// Mitsubishi GX Works2 project: 선입우선회로   PLC: Q02/Q02H

PROGRAM MAIN
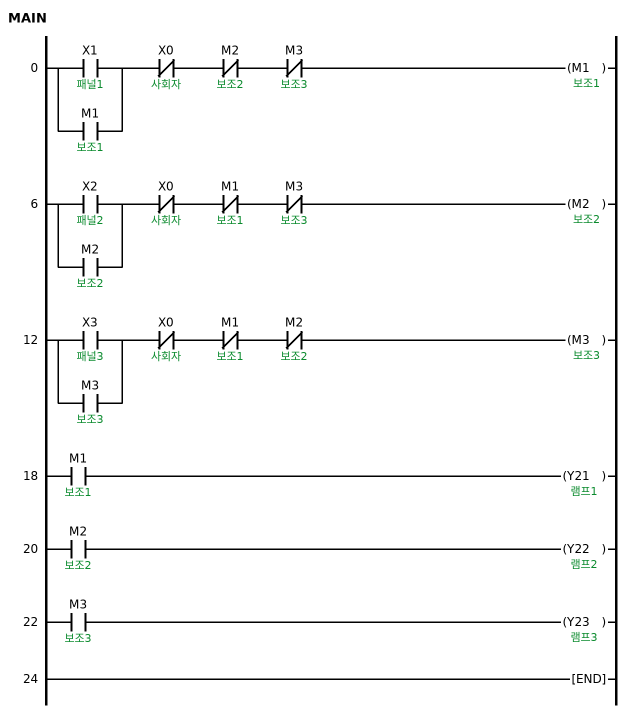
0     LD      X1  ; 패널1
      OR      M1  ; 보조1
      ANI     X0  ; 사회자
      ANI     M2  ; 보조2
      ANI     M3  ; 보조3
      OUT     M1  ; 보조1
6     LD      X2  ; 패널2
      OR      M2  ; 보조2
      ANI     X0  ; 사회자
      ANI     M1  ; 보조1
      ANI     M3  ; 보조3
      OUT     M2  ; 보조2
12    LD      X3  ; 패널3
      OR      M3  ; 보조3
      ANI     X0  ; 사회자
      ANI     M1  ; 보조1
      ANI     M2  ; 보조2
      OUT     M3  ; 보조3
18    LD      M1  ; 보조1
      OUT     Y21  ; 램프1
20    LD      M2  ; 보조2
      OUT     Y22  ; 램프2
22    LD      M3  ; 보조3
      OUT     Y23  ; 램프3
24    END
END_PROGRAM

// device comments not shown above
Y20  ; spare
M0  ; 보조0
